// Mitsubishi GX Works2 project: 3   PLC: FX3U/FX3UC

// task Task_01 (event TRUE, interval 0, priority 31): POU_01

PROGRAM POU_01
Y0 := M0 XOR M1;
END_PROGRAM
